FUNCTION_BLOCK ColorSensor (* Basic Function Block Type *)
  (* Standard: 61499-2 *)
  (* Version 0.0, 21/06/2022, Lernfabrik, WBK hackaton, Template *)
  PACKAGE Main;
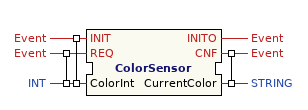
  EVENT_INPUT
    INIT WITH ColorInt; (* Initialization Request *)
    REQ WITH ColorInt; (* Normal Execution Request *)
  END_EVENT
  EVENT_OUTPUT
    INITO; (* Initialization Confirm *)
    CNF WITH CurrentColor; (* Execution Confirmation *)
  END_EVENT
  VAR_INPUT
    ColorInt : INT; (* Input event qualifier *)
  END_VAR
  VAR_OUTPUT
    CurrentColor : STRING; (* Which color is inside now? *)
  END_VAR
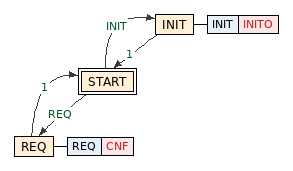
  EC_STATES
    START; (* Initial State *)
    INIT : INIT -> INITO; (* Initialization *)
    REQ : REQ -> CNF; (* Normal execution *)
  END_STATES
  EC_TRANSITIONS
    START TO INIT := INIT;
    INIT TO START := 1;
    START TO REQ := REQ;
    REQ TO START := 1;
  END_TRANSITIONS
  ALGORITHM INIT IN ST: (* Initialization algorithm *)
;
  END_ALGORITHM
  ALGORITHM REQ IN ST: (* Normally executed algorithm *)
(*BUFFER := 300;

IF ColorInt < GREENCOLOR + BUFFER AND ColorInt > BLUECOLOR - BUFFER THEN
	CurrentColor := BLUE;
END_IF; *)
;
  END_ALGORITHM
END_FUNCTION_BLOCK
